{attribute addProperty BoxType "EL2521-0000-1017"}
{attribute addProperty Id "StatusAT %I*Status_00108FF9162"}
{attribute addProperty CRC "3820918434"}
{attribute addProperty SizeInBites "16"}
{attribute addProperty SizeInBytes "2"}
TYPE PTO_Status_E3BE96A2 :
STRUCT
	{attribute addProperty Name "Status"}
	Status AT %I* : Status_00108FF9;
END_STRUCT
END_TYPE

(* stored: Version 1.2.0.0, ProductVersion 3.1.4024.9
   DUT PTO_Status_E3BE96A2: Id {7f4ba7ff-3595-48f1-aa87-af547231941a} *)
